FUNCTION Making_Toast : BOOL
VAR_INPUT
	CoffeeState : INT;
	BreadInserted : BOOL;
	LeverDown : BOOL;
END_VAR
VAR
	step : INT;
	Toasting : BOOL;
	TimerON : TON;
	JamDetected: BOOL;
END_VAR
VAR_OUTPUT
	MakingToastState : INT;
END_VAR

CASE step OF
	0 : //Idle
		IF BreadInserted AND CoffeeState = 1 THEN
			step := 10;
		END_IF
	10 : // Loading Bread
		IF LeverDown THEN
			step := 20;
		END_IF
	20 : //Toasting
		IF JamDetected THEN
			step := 0;
		ELSIF NOT JamDetected THEN
			Toasting := TRUE;
			MakingToastState := 1;
		END_IF
		TimerON(IN := Toasting, PT := T#5S);
		IF TimerON.Q THEN
			MakingToastState := 2;
			TimerON(IN := FALSE);
		END_IF
END_CASE

END_FUNCTION

(* stored: Version 1.1.0.1, ProductVersion 3.1.4024.15
   POU Making_Toast: Id {6d9288ca-62cb-465e-b746-9f270dfce14b}, SpecialFunc None *)
